// TwinCAT 3 PLC project StructuresAndFunctions
// ProgramVersion: 3.1.4023.0
// libraries:
//   Tc2_Standard, * (Beckhoff Automation GmbH)
//   Tc2_System, * (Beckhoff Automation GmbH)
//   Tc2_Utilities, * (Beckhoff Automation GmbH)
//   Tc3_Module, * (Beckhoff Automation GmbH)
//   VisuSymbols,3.5.10.0,System
// project tree:
//   DUTs/ E_EventType.TcDUT (not stored), ST_Event.TcDUT (not stored)
//   / GlobalTextList.TcGTLO (not stored), PlcTask.TcTTO
//   POUs/ Celcius_to_Fahrenet.TcPOU, Greater_Smaller.TcPOU, MAIN.TcPOU, SwapNums.TcPOU, UpdateEventTimeStampWithSystemTime.TcPOU, VisualizationManager.TcVMO (not stored)
//   VISUs/ Visualization.TcVIS (not stored)
// real-time tasks:
//   TASK PlcTask: cycle T#10ms, priority 20, ADS port 350

CONFIGURATION StructuresAndFunctions
    RESOURCE PLC ON TwinCAT3
        TASK PlcTask(INTERVAL := T#10ms, PRIORITY := 20);
        PROGRAM MAIN WITH PlcTask : MAIN;
    END_RESOURCE
END_CONFIGURATION

// ---- POUs/MAIN.TcPOU
PROGRAM MAIN
VAR
stThisIsOurFirstInstanceOfAStructure : ST_Event;
bBoolean : BOOL := FALSE;
fFahrenheit : REAL ;
nReturnGreater: INT ;
nReturnSmaller : INT;

nA : INT := 5 ;
nB : INT := 15;

END_VAR


fFahrenheit := Celcius_to_Fahrenet(fCelcius:= 5.0) ;

Greater_Smaller (nNumber1:=8,
	             nNumber2:=15,
				 nGreater => nReturnGreater,
				 nSmaller=>nReturnSmaller );			 
SwapNums(nNumber3 := nA, 
		 nNumber4 := nB);
		 
IF NOT bBoolean THEN
UpdateEventTimeStampWithSystemTime(ST_Event := stThisIsOurFirstInstanceOfAStructure);
bBoolean:= TRUE;
	
END_IF

END_PROGRAM

// ---- POUs/Celcius_to_Fahrenet.TcPOU
FUNCTION Celcius_to_Fahrenet : REAL
VAR_INPUT
	fCelcius: REAL;
	
END_VAR
VAR
END_VAR

Celcius_to_Fahrenet := fCelcius * 1.8 +32.0 ;

END_FUNCTION

// ---- POUs/Greater_Smaller.TcPOU
FUNCTION Greater_Smaller : INT
VAR_INPUT
	nNumber1 : INT;
	nNumber2 : INT;
END_VAR

VAR_OUTPUT
	nGreater : INT;
	nSmaller : INT;
	
END_VAR


IF nNumber1 > nNumber2 THEN
	nGreater := nNumber1;
	nSmaller := nNumber2;

ELSE 
	nGreater := nNumber2;
	nSmaller := nNumber1;	
END_IF

END_FUNCTION

// ---- POUs/SwapNums.TcPOU
FUNCTION SwapNums : INT
VAR_IN_OUT
nNumber3 : INT ;
nNumber4 : INT ;
	
END_VAR
VAR
	nNumberTemp : INT;
	
END_VAR


nNumberTemp := nNumber3;
nNumber3 := nNumber4;
nNumber4 := nNumberTemp;

END_FUNCTION

// ---- POUs/UpdateEventTimeStampWithSystemTime.TcPOU
FUNCTION UpdateEventTimeStampWithSystemTime 
VAR_INPUT
	ST_Event:  REFERENCE TO ST_Event;
END_VAR
VAR
	FbGETSYSTEMTIME : GETSYSTEMTIME; // Bu FONKSİYON BİZE sistem zamanını veriyor.

	st_FILETIME : T_FILETIME; // Bu structa saklıyoruz sistemden çektiğimiz saati. Çünkü biz DATE TIME döüştürmemiz grekiyor bunun için de önce FILETIME kaydettik buradan dönüştürecez.

END_VAR

FbGETSYSTEMTIME(timeLoDW => st_FILETIME.dwLowDateTime,
	            timeHiDW => st_FILETIME.dwHighDateTime);
				
	ST_Event.dtTimestamp:= FILETIME_TO_DT(fileTime := st_FILETIME);

END_FUNCTION
